Fanuc KAREL source: kd00055.KL

-- PROVISIONAL review KL for V940-1; original PC SHA256 c2b79753a0f6783e661c32afdd0996d8b69b6624973ade41637492126010c6f6
-- Incomplete behavior may be omitted. Consult companion uncertainty JSON. Do not deploy.
PROGRAM KD00055
%NOLOCKGROUP
VAR
  I : INTEGER
  J : INTEGER
  B : BOOLEAN
  R : REAL
  S : STRING[80]
BEGIN
  -- V9_ZERO_TABLE_METADATA_HINT layout=0001; no indexed target words; source/name/runtime held
  -- UNRESOLVED_PC offsets 5-25; opcodes 9D,81,18,9D,1B,9D,12,2E,1B,9D,13,04
  -- UNRESOLVED_PC offsets 30-34; opcodes 7F
END KD00055
